(* PLC project Tc2_Utilities.F_WORD Demo, tc3-libraries-kb TwinCAT 3.1 *)
(* stored: creationDateTime 2026-05-10T14:00:00, modificationDateTime 2026-05-10T14:00:00 *)

PROGRAM P_Demo_F_WORD
  VAR
    rResult : T_Arg;  (* F_WORD 返回值 *)
    bRun : BOOL;  (* 触发一次调用 *)
    v : WORD;  (* 测试用本地变量 *)
  END_VAR

            // ============================================================
// Tc2_Utilities.F_WORD 演示程序（FUNCTION）
// ============================================================
// 验证步骤：
//   1. 引用 Tc2_Utilities
//   2. 编译 + 登录
//   3. 强制 bRun := TRUE 一个周期
//   4. 观察 rResult 应为 ...
// ============================================================

IF bRun THEN
    rResult := F_WORD(in := v);
    bRun := FALSE;
END_IF;

          
END_PROGRAM
